(* IEC 61131-3 sources: beckhoffAutomationInterface/ST/Shark/Lib/Controllers/Interfaces, 3 files *)

(* ---- ST_ControllerStatus.st ---- *)
(* Consolidated status structure for controllers. *)
TYPE ST_ControllerStatus :
STRUCT
    // Process Values
    rMeasuredValue      : LREAL;             // Current measurement
    rSetpoint           : LREAL;             // Active setpoint
    rOutput             : LREAL;             // Control output (0-100% or similar)
    // State Flags
    bEnabled            : BOOL;              // Operation enabled
    bAtSetpoint         : BOOL;              // Within tolerance
    bSafetyTripped      : BOOL;              // TRUE when a safety interlock has latched (heater forced OFF)
    // Diagnostics
    stError             : ST_Error;          // Active error details
END_STRUCT
END_TYPE

(* ---- I_Controller.st ---- *)
(* Base Controller Interface. Defines core functionality common to all controller types. *)
INTERFACE I_Controller EXTENDS __System.IQueryInterface

METHOD Enable : BOOL
VAR_INPUT
    bEnable : BOOL;
END_VAR
END_METHOD

METHOD SetSetpoint : BOOL
VAR_INPUT
    rDesiredSetpoint : LREAL;
END_VAR
END_METHOD

METHOD GetStatus : ST_ControllerStatus
END_METHOD

METHOD Reset : BOOL
END_METHOD

END_INTERFACE

(* ---- I_Tunable.st ---- *)
(* Tunable controller interface.

A tunable is a controller that, in addition to the normal I_Controller surface
(Enable / SetSetpoint / GetStatus / Reset), supports switching its control mode
at runtime — most importantly into the Beckhoff PID self-tuning (autotune) mode.

Implemented by both a single channel (FB_BeckhoffTempController) and a whole
heat zone (FB_HeatZone). A zone cascades the mode to every channel it owns, so
the same panel can tune one channel or an entire zone interchangeably
(Liskov substitution). *)
INTERFACE I_Tunable EXTENDS I_Controller

(* Switch the controller (or every channel of a zone) into the given control
   mode, e.g. E_CTRL_MODE.eCTRL_MODE_TUNE to start autotuning or
   E_CTRL_MODE.eCTRL_MODE_ACTIVE to return to normal closed-loop control. *)
METHOD SetControlMode : BOOL
VAR_INPUT
    eMode : E_CTRL_MODE;
END_VAR
END_METHOD

(* Current control mode (for a zone: the last mode commanded to its channels). *)
METHOD GetControlMode : E_CTRL_MODE
END_METHOD

END_INTERFACE
